/// Enumeration of possible axis gear modes.
TYPE E_GearMode :
(
	/// Gear mode not set
	eGearMode_none := 0,
	/// Gear in
	eGearMode_in,
	/// Gear out
	eGearMode_out
);
END_TYPE

(* stored: Version 1.1.0.1, ProductVersion 3.1.4022.9
   DUT E_GearMode: Id {aa1816ba-df28-4e85-a2c8-b7fdbaa6a002} *)
